TYPE ST_SoftSettings_DcLink :
STRUCT
		b_Enable 			: BOOL;
END_STRUCT
END_TYPE

(* stored: Version 1.1.0.1, ProductVersion 3.1.4026.18
   DUT ST_SoftSettings_DcLink: Id {b8c31f81-6180-4b4c-9f9b-30c18bc2a326} *)
